// Mitsubishi GX Works2 project: 0715MCMCR2   PLC: Q02/Q02H

PROGRAM MAIN
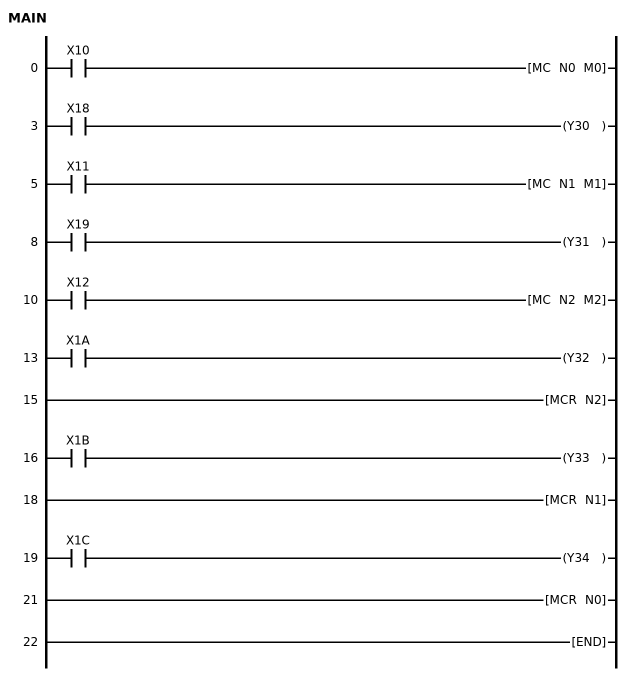
0     LD      X10
      MC      N0 M0
3     LD      X18
      OUT     Y30
5     LD      X11
      MC      N1 M1
8     LD      X19
      OUT     Y31
10    LD      X12
      MC      N2 M2
13    LD      X1A
      OUT     Y32
15    MCR     N2
16    LD      X1B
      OUT     Y33
18    MCR     N1
19    LD      X1C
      OUT     Y34
21    MCR     N0
22    END
END_PROGRAM
